(* IEC 61131-3 sources: axopen.templates/axopen.template.simple/ax/src/templates/starterunit/Data, 2 files *)

(* ---- ProcessDataPayload.st ---- *)
NAMESPACE axosimple.StarterUnitTemplate
    USING axosimple;
    USING AXOpen.Data;
    USING AXOpen.Core;
    USING System.Strings;

    {S7.extern=ReadWrite}
    CLASS ProcessDataPayload
        EXTENDS AXOpen.Data.AxoDataEntity
        VAR PUBLIC
            CounterDelay : ULINT;

            PartPresence        : AXOpen.Inspectors.AxoDigitalInspector;
            JigDataMatrixCode   : AXOpen.Inspectors.AxoDataInspector;
            LoadPosition        : AXOpen.Inspectors.AxoAnalogueInspector;
        END_VAR
    END_CLASS
END_NAMESPACE

(* ---- TechnologyDataPayload.st ---- *)
NAMESPACE axosimple.StarterUnitTemplate
    USING axosimple;
    USING AXOpen.Data;
    USING AXOpen.Core;
    USING System.Strings;

    {S7.extern=ReadWrite}
    CLASS TechnologyDataPayload
        EXTENDS AXOpen.Data.AxoDataEntity
        VAR PUBLIC

            Header : axosimple.TechnologyUnitHeader;

            HeatingTemperature   : REAL;

        END_VAR
    END_CLASS
END_NAMESPACE
